Staubli VAL3: start.pgx

program start()
begin
  movej(jAproachPiece,tTool,mNomSpeed)
  waitEndMove()
  movel(pGetObject,tTool,mNomSpeed)
  waitEndMove()
  close(tTool)
  waitEndMove()
  movej(jAproachPiece,tTool,mNomSpeed)
  waitEndMove()

end
